INTERFACE I_Humano

METHOD Correr
VAR_INPUT
END_VAR
END_METHOD

PROPERTY Nombre : STRING
GET
END_GET
SET
END_SET
END_PROPERTY

END_INTERFACE

(* stored: Version 1.1.0.1, ProductVersion 3.1.4024.12
   Itf I_Humano: Id {98075f32-8b2f-4edb-a073-71d3efcc29ac}
   Method Correr: Id {4cc6fa0e-9db5-4ae9-a122-04ea480348ac}
   Property Nombre: Id {89534d93-73f5-46a3-8e7f-76e7fc424d65}
   Get Get: Id {299b0a8d-6f62-4b1d-aba1-1f8f526f17d4}
   Set Set: Id {81c806db-db62-4cce-84aa-677c40aa1d1a} *)
